// TIA Portal V20 export
FUNCTION_BLOCK "FB_Nouveau"   // FB91, SCL
{ S7_Optimized_Access := 'TRUE' }
// stored: MemoryReserve 100, SetENOAutomatically false
   VAR
      "#sExtLoadUnloadTimer1" : TON_TIME;
      "#sExtLoadUnloadTimer2" { S7_SetPoint := 'True'} : TON_TIME;
   END_VAR
BEGIN
   REGION Ext Load/Unload Time
       // Necessaire pour Dry Run
       // #sExtLoadUnloadTimer1(IN := "DB_LoaderShuttle1".sExtLoadUnload.sCurrent_Step_NB = 50
       //                       OR "DB_LoaderShuttle1".sExtLoadUnload.sCurrent_Step_NB = 80
       //                       OR "DB_LoaderShuttle1".sExtLoadUnload.sCurrent_Step_NB = 110,
       //                       PT := t#3s);
       // "DB_SonplasMain".sSonplasLoader.iPartInShuttle1Finished := #sExtLoadUnloadTimer1.Q;

       // #sExtLoadUnloadTimer2(IN := "DB_LoaderShuttle2".sExtLoadUnload.sCurrent_Step_NB = 50
       //                       OR "DB_LoaderShuttle2".sExtLoadUnload.sCurrent_Step_NB = 80
       //                       OR "DB_LoaderShuttle2".sExtLoadUnload.sCurrent_Step_NB = 110,
       //                       PT := t#3s);
       // "DB_SonplasMain".sSonplasLoader.iPartInShuttle2Finished := #sExtLoadUnloadTimer2.Q;
   END_REGION
END_FUNCTION_BLOCK
